Universal Robots PolyScope program: set_b_draw_borders.bak.urp

Program set_b_draw_borders.bak (installation=default directory=/programs createdIn=5.11.9.1010452 lastSavedIn=5.11.9.1010452 robotSerialNumber=20225200364)
Calibrated DH parameters: a=[0.00002, -0.569483, -0.54992, -0.00001, -0.000036, 0]; d=[0.180894, -146.691669, 192.918669, -46.053088, 0.119778, 0.115602]; alpha=[1.571425, -0.001534, 0.003359, 1.568739, -1.571477, 0]; deltaTheta=[0, 0.376258, -0.101074, -0.275185, -0.000002, 0]
Robot Program (runOnlyOnce=true)
  Script file /programs/usbdisk/draw_borders.script
    | def Machining3():
    |   # Default parameters:
    |   global speed_ms = 0.3
    |   global speed_rads = 0.75
    |   global accel_mss = 3
    |   global accel_radss = 1.2
    |   global blend_radius_m = 0.001
    | 
    |   # Add subprograms here
    |   # Start of main program
    |   # Program generated by RoboDK v5.6.5 for UR10e on 17/10/2023 11:41:04
    |   # Using nominal kinematics.
    |   blend_radius_m = 0.001
    |   speed_ms = 1.000
    |   # set_reference(p[0.335000, -0.154000, -0.015800, 0.000000, 0.000000, 0.000000])
    |   set_tcp(p[0.000000, 0.000000, 0.252000, 0.000000, 0.000000, 0.000000])
    |   # Show Tool
    |   movej([0.061043, -1.073805, -2.582860, -1.055724, 1.570796, 1.631840],accel_radss,speed_rads,0,blend_radius_m)
    |   movel([0.061043, -1.164815, -2.648932, -0.898642, 1.570796, 1.631840],accel_mss,speed_ms,0,blend_radius_m)
    |   speed_ms = 1.000
    |   speed_ms = 0.005
    |   movel([0.061043, -1.124589, -2.623317, -0.964483, 1.570796, 1.631840],accel_mss,speed_ms,0,blend_radius_m)
    |   speed_ms = 1.000
    |   movel([0.061043, -1.164815, -2.648932, -0.898642, 1.570796, 1.631840],accel_mss,speed_ms,0,blend_radius_m)
    |   speed_ms = 0.040
    |   speed_ms = 1.000
    |   movel([0.157276, -1.127729, -2.665258, -0.919402, 1.570796, 1.728073],accel_mss,speed_ms,0,blend_radius_m)
    |   speed_ms = 0.005
    |   movel([0.157276, -1.174031, -2.690432, -0.847927, 1.570796, 1.728073],accel_mss,speed_ms,0,blend_radius_m)
    |   speed_ms = 0.035
    |   movel([0.061043, -1.210716, -2.673294, -0.828379, 1.570796, 1.631840],accel_mss,speed_ms,0,blend_radius_m)
    |   movel([0.051500, -1.358795, -2.587796, -0.765798, 1.570796, 1.622297],accel_mss,speed_ms,0,blend_radius_m)
    |   movel([0.044558, -1.480296, -2.495031, -0.737062, 1.570796, 1.615354],accel_mss,speed_ms,0,blend_radius_m)
    |   movel([0.113774, -1.462570, -2.509956, -0.739863, 1.570796, 1.684571],accel_mss,speed_ms,0,blend_radius_m)
    |   movel([0.183803, -1.448210, -2.521691, -0.742489, 1.570796, 1.754599],accel_mss,speed_ms,0,blend_radius_m)
    |   movel([0.213690, -1.314067, -2.616588, -0.781734, 1.570796, 1.784487],accel_mss,speed_ms,0,blend_radius_m)
    |   movel([0.255784, -1.142912, -2.703858, -0.865619, 1.570796, 1.826580],accel_mss,speed_ms,0,blend_radius_m)
    |   movel([0.157276, -1.174031, -2.690432, -0.847927, 1.570796, 1.728073],accel_mss,speed_ms,0,blend_radius_m)
    |   movel([0.154107, -1.175144, -2.689933, -0.847312, 1.570796, 1.724904],accel_mss,speed_ms,0,blend_radius_m)
    |   speed_ms = 0.005
    |   movel([0.154107, -1.128851, -2.664784, -0.918754, 1.570796, 1.724904],accel_mss,speed_ms,0,blend_radius_m)
    |   speed_ms = 1.000
    |   movel([0.154107, -1.038314, -2.596953, -1.077123, 1.570796, 1.724904],accel_mss,speed_ms,0,blend_radius_m)
    |   # End of main program
    | end
    | 
    | Machining3()
